// TIA Portal V18 export
// export: Created 2026-01-09T11:32:05.6336649Z, ExportSetting WithDefaults, DisplayName Totally Integrated Automation Portal, DisplayVersion V18 Update 5, DisplayName TIA Portal Openness, DisplayVersion V18 Update 5, DisplayName TIA Portal Teamcenter Gateway, DisplayVersion V18, DisplayName TIA Portal Version Control Interface, DisplayVersion V18, DisplayName SINAMICS Startdrive Advanced, DisplayVersion V18 SP2 Update 1, DisplayName SINAMICS Startdrive G110M, G120, G120C, G120D, G120P, G115D, DisplayVersion V18 SP2 Update 1, DisplayName SINAMICS Startdrive G130, G150, S120, S150, SINAMICS MV, S210, G220, S200, DisplayVersion V18 SP2 Update 1, DisplayName STEP 7 Professional, DisplayVersion V18 Update 5, DisplayName STEP 7 Safety, DisplayVersion V18, DisplayName WinCC Professional, DisplayVersion V18 Update 5
TagTable "弹窗"
  Win101 : Int  (PLC tag ST10_GeneralData.HMI.Win.10x弹窗[1], CPU S71500-2PN_TP700, 100 ms)
  Win102 : Int  (PLC tag ST10_GeneralData.HMI.Win.10x弹窗[2], CPU S71500-2PN_TP700, 100 ms)
  Win103 : Int  (PLC tag ST10_GeneralData.HMI.Win.10x弹窗[3], CPU S71500-2PN_TP700, 100 ms)
  Win104 : Int  (PLC tag ST10_GeneralData.HMI.Win.10x弹窗[4], CPU S71500-2PN_TP700, 100 ms)
  Win105 : Int  (PLC tag ST10_GeneralData.HMI.Win.10x弹窗[5], CPU S71500-2PN_TP700, 100 ms)
  Win106 : Int  (PLC tag ST10_GeneralData.HMI.Win.10x弹窗[6], CPU S71500-2PN_TP700, 100 ms)
  Win107 : Int  (PLC tag ST10_GeneralData.HMI.Win.10x弹窗[7], CPU S71500-2PN_TP700, 100 ms)
  Win108 : Int  (PLC tag ST10_GeneralData.HMI.Win.10x弹窗[8], CPU S71500-2PN_TP700, 100 ms)
  Win109 : Int  (PLC tag ST10_GeneralData.HMI.Win.10x弹窗[9], CPU S71500-2PN_TP700, 100 ms)
  Win110 : Int  (PLC tag ST10_GeneralData.HMI.Win.10x弹窗[10], CPU S71500-2PN_TP700, 100 ms)
  Win201 : Int  (PLC tag ST10_GeneralData.HMI.Win.20x弹窗[1], CPU S71500-2PN_TP700, 100 ms)
  Win202 : Int  (PLC tag ST10_GeneralData.HMI.Win.20x弹窗[2], CPU S71500-2PN_TP700, 100 ms)
  Win203 : Int  (PLC tag ST10_GeneralData.HMI.Win.20x弹窗[3], CPU S71500-2PN_TP700, 100 ms)
  Win204 : Int  (PLC tag ST10_GeneralData.HMI.Win.20x弹窗[4], CPU S71500-2PN_TP700, 100 ms)
  Win205 : Int  (PLC tag ST10_GeneralData.HMI.Win.20x弹窗[5], CPU S71500-2PN_TP700, 100 ms)
  Win206 : Int  (PLC tag ST10_GeneralData.HMI.Win.20x弹窗[6], CPU S71500-2PN_TP700, 100 ms)
  Win207 : Int  (PLC tag ST10_GeneralData.HMI.Win.20x弹窗[7], CPU S71500-2PN_TP700, 100 ms)
  Win208 : Int  (PLC tag ST10_GeneralData.HMI.Win.20x弹窗[8], CPU S71500-2PN_TP700, 100 ms)
  Win209 : Int  (PLC tag ST10_GeneralData.HMI.Win.20x弹窗[9], CPU S71500-2PN_TP700, 100 ms)
  Win210 : Int  (PLC tag ST10_GeneralData.HMI.Win.20x弹窗[10], CPU S71500-2PN_TP700, 100 ms)
  Win301 : Int  (PLC tag ST10_GeneralData.HMI.Win.30x弹窗[1], CPU S71500-2PN_TP700, 100 ms)
  Win302 : Int  (PLC tag ST10_GeneralData.HMI.Win.30x弹窗[2], CPU S71500-2PN_TP700, 100 ms)
  Win303 : Int  (PLC tag ST10_GeneralData.HMI.Win.30x弹窗[3], CPU S71500-2PN_TP700, 100 ms)
  Win304 : Int  (PLC tag ST10_GeneralData.HMI.Win.30x弹窗[4], CPU S71500-2PN_TP700, 100 ms)
  Win305 : Int  (PLC tag ST10_GeneralData.HMI.Win.30x弹窗[5], CPU S71500-2PN_TP700, 100 ms)
  Win306 : Int  (PLC tag ST10_GeneralData.HMI.Win.30x弹窗[6], CPU S71500-2PN_TP700, 100 ms)
  Win307 : Int  (PLC tag ST10_GeneralData.HMI.Win.30x弹窗[7], CPU S71500-2PN_TP700, 100 ms)
  Win308 : Int  (PLC tag ST10_GeneralData.HMI.Win.30x弹窗[8], CPU S71500-2PN_TP700, 100 ms)
  Win309 : Int  (PLC tag ST10_GeneralData.HMI.Win.30x弹窗[9], CPU S71500-2PN_TP700, 100 ms)
  Win310 : Int  (PLC tag ST10_GeneralData.HMI.Win.30x弹窗[10], CPU S71500-2PN_TP700, 100 ms)
  Win401 : Int  (PLC tag ST10_GeneralData.HMI.Win.40x弹窗[1], CPU S71500-2PN_TP700, 100 ms)
  Win402 : Int  (PLC tag ST10_GeneralData.HMI.Win.40x弹窗[2], CPU S71500-2PN_TP700, 100 ms)
  Win403 : Int  (PLC tag ST10_GeneralData.HMI.Win.40x弹窗[3], CPU S71500-2PN_TP700, 100 ms)
  Win404 : Int  (PLC tag ST10_GeneralData.HMI.Win.40x弹窗[4], CPU S71500-2PN_TP700, 100 ms)
  Win405 : Int  (PLC tag ST10_GeneralData.HMI.Win.40x弹窗[5], CPU S71500-2PN_TP700, 100 ms)
  Win406 : Int  (PLC tag ST10_GeneralData.HMI.Win.40x弹窗[6], CPU S71500-2PN_TP700, 100 ms)
  Win407 : Int  (PLC tag ST10_GeneralData.HMI.Win.40x弹窗[7], CPU S71500-2PN_TP700, 100 ms)
  Win408 : Int  (PLC tag ST10_GeneralData.HMI.Win.40x弹窗[8], CPU S71500-2PN_TP700, 100 ms)
  Win409 : Int  (PLC tag ST10_GeneralData.HMI.Win.40x弹窗[9], CPU S71500-2PN_TP700, 100 ms)
  Win410 : Int  (PLC tag ST10_GeneralData.HMI.Win.40x弹窗[10], CPU S71500-2PN_TP700, 100 ms)
  Win : Int  (PLC tag ST10_GeneralData.HMI.Win.Win, CPU S71500-2PN_TP700, 100 ms)
  WinBuffer : Int  (PLC tag ST10_GeneralData.HMI.Win.WinBullfer, CPU S71500-2PN_TP700, 100 ms)
